PROGRAM MAIN
VAR
	fbSensor1		: FB_PT100;
	fbMotor1		: FB_Motor(TempSensor := fbSensor1);
	fbSensor2		: FB_PT1000;
	fbMotor2		: FB_Motor(fbSensor2);
END_VAR

// Motors
fbSensor1();
fbMotor1();	
fbSensor2();
fbMotor2();

END_PROGRAM

(* stored: Version 1.1.0.1, ProductVersion 3.1.4022.18
   POU MAIN: Id {4397753d-6707-4ee1-9ec6-9f41f8444ae4}, SpecialFunc None *)
